// TIA Portal V20 export
DATA_BLOCK "DB_Scanner"   // DB128
// stored: InstanceOfName FB_Scanner, InstanceOfType FB
"FB_Scanner"
   // VAR
   //    sScannerComm : "FB_ScannerComm";
   //    sReadR_Param { S7_SetPoint := 'True'} : "LBP_ReadVar";
   //    sWriteR_Param { S7_SetPoint := 'True'} : "LBP_WriteVar";
   //    sError { ExternalAccessible := 'False'; ExternalVisible := 'False'; ExternalWritable := 'False'} : Bool;
   //    sNDR { ExternalAccessible := 'False'; ExternalVisible := 'False'; ExternalWritable := 'False'} : Bool;
   //    sState { ExternalAccessible := 'False'; ExternalVisible := 'False'; ExternalWritable := 'False'} : Word;
   //    sR94 : LReal;
   //    sR95 : LReal;
   //    sR96 : LReal;
   //    sR97 : LReal;
   //    sJobNamePart : DInt;
   //    sJobNamePowerMeter : DInt;
   //    sMeasureZ : LReal;
   //    sVarName { S7_SetPoint := 'True'} : String;
   //    sReadGUD_JobNamePart { S7_SetPoint := 'True'} : "LBP_ReadGUD";
   //    sReadGUD_JobNamePowerMeter { S7_SetPoint := 'True'} : "LBP_ReadGUD";
   //    sReadGUD_MeasureZ { S7_SetPoint := 'True'} : "LBP_ReadGUD";
   //    sWriteR_ParamReq { S7_SetPoint := 'True'} : Bool;
   //    sTimePulseWriteParam : TON_TIME;
   // END_VAR
BEGIN
END_DATA_BLOCK
